INTERFACE I_Header

METHOD PUBLIC ToString
VAR_INPUT
	Destination : REFERENCE TO STRING(ServerConfiguration.HEADER_STRING_SIZE);
END_VAR
END_METHOD

METHOD PUBLIC TryGetField : BOOL;
VAR_INPUT
	Key : STRING;
	Destination : ANY;
END_VAR
END_METHOD

METHOD PUBLIC TryWriteField : BOOL;
VAR_INPUT
	Key : STRING;
	Source : ANY;
END_VAR
END_METHOD

END_INTERFACE

(* stored: Version 1.1.0.1, ProductVersion 3.1.4024.12
   Itf I_Header: Id {04632699-d748-00ea-1005-f5546e3f6c1e}
   Method ToString: Id {566f8047-311a-029d-33db-a82b9e876b85}
   Method TryGetField: Id {e70db9ed-36d4-0ada-1a85-de539c3373c3}
   Method TryWriteField: Id {25401a29-f0c9-0732-33fe-e36f90f78706} *)
